Fanuc KAREL source: kt00134.KL

-- PROVISIONAL review KL for V770-1; original PC SHA256 9c4620db7bea28dac2ed8bcb1470d119f2addf28eaffdf1a96eda3967805fc4c
-- Incomplete behavior may be omitted. Consult companion uncertainty JSON. Do not deploy.
PROGRAM KT00134
%NOLOCKGROUP
VAR
  I1 : INTEGER
  OUT : REAL
-- UNRESOLVED_DECL Y2 type=002018
BEGIN
  -- UNRESOLVED_PC offsets 5-16; opcodes 2E,23
  -- UNRESOLVED_PC offsets 21-35; opcodes 2E,22,9D,33,B2
  -- UNRESOLVED_PC offsets 40-63; opcodes 21,22,9D,33,B1,55,64,23
  -- UNRESOLVED_PC offsets 68-72; opcodes 7F
END KT00134
